FUNCTION F_PointInnerRect : BOOL
VAR_INPUT
	stPoint		: ST_3DPoint;
	stRectangle : ST_Rectangle;
END_VAR
VAR
END_VAR

F_PointInnerRect := (stPoint.X >= stRectAngle.X1) AND
					(stPoint.X <= stRectAngle.X2) AND
					(stPoint.Y >= stRectAngle.Y1) AND
					(stPoint.Y <= stRectAngle.Y2);

END_FUNCTION

(* stored: Version 1.1.0.1, ProductVersion 3.1.4020.12
   POU F_PointInnerRect: Id {be2359e1-0790-45a5-943e-26be1bcfc302}, SpecialFunc None *)
